// TIA Portal V20 export
DATA_BLOCK "AdjFast"   // DB506
{ S7_Optimized_Access := 'TRUE'; DB_Accessible_From_OPC_UA := 'FALSE' }
// stored: AutoNumber false, DBAccessibleFromOPCUA false, MemoryReserve 100
   VAR
      Top { ExternalAccessible := 'False'; ExternalVisible := 'False'; ExternalWritable := 'False'} : Struct   // adjustment top
         Mode : Int := 0;   // 1=VAI / 2=SIN VA / 3=Bestehorn VAJ
         Test : Struct
            ModeActive : Bool := false;   // mode test active (move between testpos 1 and 2)
            TarPos : Real := 5.0;   // target positon [mm]
            TarPos1 : Real := 5.0;   // target positon 1 [mm]
            TarPos2 : Real := 155.0;   // target positon 2 [mm]
            TimePosOk : Time := T#2s;   // time for position ok to switch to other position
         END_STRUCT;
         VAI : Struct
            Par1 : Real := 50.0;   // target positon [mm]
            Par2 : Real := 2.0;   // maximal velocity [m/s]
            Par3 : Real := 12.0;   // acceleration [m/s²]
            Par4 : Real := 12.0;   // deceleration [m/s²]
         END_STRUCT;
         SinVA : Struct
            Par1 : Real := 50.0;   // target positon [mm]
            Par2 : Real := 2.0;   // maximal velocity [m/s]
            Par3 : Real := 18.0;   // maixmal acceleration/deceleration [m/s²]
            Par4 : Real := 0.0;   // not used
         END_STRUCT;
         BestehornVAJ : Struct
            Par1 : Real := 50.0;   // target positon [mm]
            Par2 : Real := 2.0;   // maximal velocity [m/s]
            Par3 : Real := 24.0;   // maixmal acceleration/deceleration [m/s²]
            Par4 : Real := 450.0;   // maximal jerk [m/s³]
         END_STRUCT;
         Current : Struct   // current monitoring
            Man : Struct   // manual mode
               War : Struct
                  MinValue : Real := -3.0;   // min current value
                  MaxValue : Real := 2.0;   // max current value
                  Err : Bool;   // warning error
               END_STRUCT;
               Err : Struct
                  MinValue : Real := -3.0;   // min current value
                  MaxValue : Real := 2.0;   // max current value
                  Err : Bool;   // error
               END_STRUCT;
            END_STRUCT;
            Auto : Struct   // auto mode
               War : Struct
                  MinValue : Real := -15.0;   // min current value
                  MaxValue : Real := 16.0;   // max current value
                  Err : Bool;   // warning error
               END_STRUCT;
               Err : Struct
                  MinValue : Real := -15.0;   // min current value
                  MaxValue : Real := 16.0;   // max current value
                  Err : Bool;   // error
               END_STRUCT;
            END_STRUCT;
         END_STRUCT;
      END_STRUCT;
      Left { ExternalAccessible := 'False'; ExternalVisible := 'False'; ExternalWritable := 'False'} : Struct   // adjustment left
         Mode : Int := 0;   // 1=VAI / 2=SIN VA / 3=Bestehorn VAJ
         Test : Struct
            ModeActive : Bool := false;   // mode test active (move between testpos 1 and 2)
            TarPos : Real := 5.0;   // target positon [mm]
            TarPos1 : Real := 5.0;   // target positon 1 [mm]
            TarPos2 : Real := 155.0;   // target positon 2 [mm]
            TimePosOk : Time := T#2s;   // time for position ok to switch to other position
         END_STRUCT;
         VAI : Struct
            Par1 : Real := 50.0;   // target positon [mm]
            Par2 : Real := 2.0;   // maximal velocity [m/s]
            Par3 : Real := 12.0;   // acceleration [m/s²]
            Par4 : Real := 12.0;   // deceleration [m/s²]
         END_STRUCT;
         SinVA : Struct
            Par1 : Real := 50.0;   // target positon [mm]
            Par2 : Real := 2.0;   // maximal velocity [m/s]
            Par3 : Real := 18.0;   // maixmal acceleration/deceleration [m/s²]
            Par4 : Real := 0.0;   // not used
         END_STRUCT;
         BestehornVAJ : Struct
            Par1 : Real := 50.0;   // target positon [mm]
            Par2 : Real := 2.0;   // maximal velocity [m/s]
            Par3 : Real := 24.0;   // maixmal acceleration/deceleration [m/s²]
            Par4 : Real := 450.0;   // maximal jerk [m/s³]
         END_STRUCT;
         Current : Struct   // current monitoring
            Man : Struct   // manual mode
               War : Struct
                  MinValue : Real := -3.0;   // min current value
                  MaxValue : Real := 2.0;   // max current value
                  Err : Bool;   // warning error
               END_STRUCT;
               Err : Struct
                  MinValue : Real := -3.0;   // min current value
                  MaxValue : Real := 2.0;   // max current value
                  Err : Bool;   // error
               END_STRUCT;
            END_STRUCT;
            Auto : Struct   // auto mode
               War : Struct
                  MinValue : Real := -15.0;   // min current value
                  MaxValue : Real := 16.0;   // max current value
                  Err : Bool;   // warning error
               END_STRUCT;
               Err : Struct
                  MinValue : Real := -15.0;   // min current value
                  MaxValue : Real := 16.0;   // max current value
                  Err : Bool;   // error
               END_STRUCT;
            END_STRUCT;
         END_STRUCT;
      END_STRUCT;
      Right { ExternalAccessible := 'False'; ExternalVisible := 'False'; ExternalWritable := 'False'} : Struct   // adjustment right
         Mode : Int := 0;   // 1=VAI / 2=SIN VA / 3=Bestehorn VAJ
         Test : Struct
            ModeActive : Bool := false;   // mode test active (move between testpos 1 and 2)
            TarPos : Real := 5.0;   // target positon [mm]
            TarPos1 : Real := 5.0;   // target positon 1 [mm]
            TarPos2 : Real := 155.0;   // target positon 2 [mm]
            TimePosOk : Time := T#2s;   // time for position ok to switch to other position
         END_STRUCT;
         VAI : Struct
            Par1 : Real := 50.0;   // target positon [mm]
            Par2 : Real := 2.0;   // maximal velocity [m/s]
            Par3 : Real := 12.0;   // acceleration [m/s²]
            Par4 : Real := 12.0;   // deceleration [m/s²]
         END_STRUCT;
         SinVA : Struct
            Par1 : Real := 50.0;   // target positon [mm]
            Par2 : Real := 2.0;   // maximal velocity [m/s]
            Par3 : Real := 18.0;   // maixmal acceleration/deceleration [m/s²]
            Par4 : Real := 0.0;   // not used
         END_STRUCT;
         BestehornVAJ : Struct
            Par1 : Real := 50.0;   // target positon [mm]
            Par2 : Real := 2.0;   // maximal velocity [m/s]
            Par3 : Real := 24.0;   // maixmal acceleration/deceleration [m/s²]
            Par4 : Real := 450.0;   // maximal jerk [m/s³]
         END_STRUCT;
         Current : Struct   // current monitoring
            Man : Struct   // manual mode
               War : Struct
                  MinValue : Real := -3.0;   // min current value
                  MaxValue : Real := 2.0;   // max current value
                  Err : Bool;   // warning error
               END_STRUCT;
               Err : Struct
                  MinValue : Real := -3.0;   // min current value
                  MaxValue : Real := 2.0;   // max current value
                  Err : Bool;   // error
               END_STRUCT;
            END_STRUCT;
            Auto : Struct   // auto mode
               War : Struct
                  MinValue : Real := -15.0;   // min current value
                  MaxValue : Real := 16.0;   // max current value
                  Err : Bool;   // warning error
               END_STRUCT;
               Err : Struct
                  MinValue : Real := -15.0;   // min current value
                  MaxValue : Real := 16.0;   // max current value
                  Err : Bool;   // error
               END_STRUCT;
            END_STRUCT;
         END_STRUCT;
      END_STRUCT;
   END_VAR
BEGIN
END_DATA_BLOCK
